PROGRAM F_FIN_CICLO
VAR_INPUT

	Func:E_funcio;
END_VAR
VAR
	///Activa
	xActv: BOOL;
	xA_FIN_CICLO: BOOL;
END_VAR

	
(* 10 Fin de ciclo*)

xActv:=func.Actv_Funcio;
ATL.PE.xEndBatch := xActv; 

(* Alarma Fin de Ciclo *)
xA_FIN_CICLO := xActv  ;

END_PROGRAM

(* stored: Version 1.1.0.1, ProductVersion 3.1.4024.10
   POU F_FIN_CICLO: Id {42483825-9c47-42bd-9808-7018f31193ad}, SpecialFunc None *)
